// Mitsubishi GX Works2 project: plc 기말 신호등   PLC: Q02/Q02H

PROGRAM MAIN
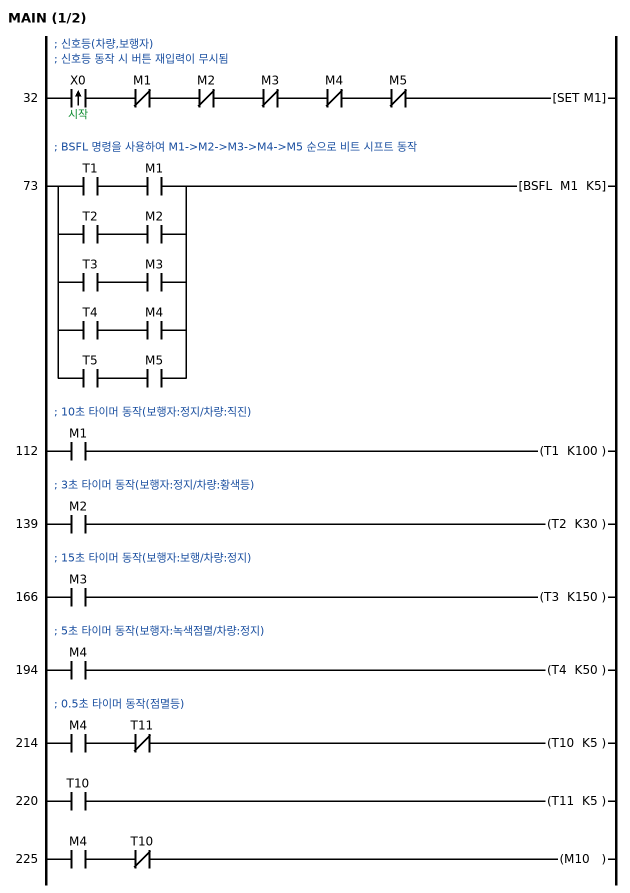
; 신호등(차량,보행자)
; 신호등 동작 시 버튼 재입력이 무시됨
32    LDP     X0  ; 시작
      ANI     M1
      ANI     M2
      ANI     M3
      ANI     M4
      ANI     M5
      SET     M1
; BSFL 명령을 사용하여 M1->M2->M3->M4->M5 순으로 비트 시프트 동작
73    LD      T1
      AND     M1
      LD      T2
      AND     M2
      ORB
      LD      T3
      AND     M3
      ORB
      LD      T4
      AND     M4
      ORB
      LD      T5
      AND     M5
      ORB
      BSFL    M1 K5
; 10초 타이머 동작(보행자:정지/차량:직진)
112   LD      M1
      OUT     T1 K100
; 3초 타이머 동작(보행자:정지/차량:황색등)
139   LD      M2
      OUT     T2 K30
; 15초 타이머 동작(보행자:보행/차량:정지)
166   LD      M3
      OUT     T3 K150
; 5초 타이머 동작(보행자:녹색점멸/차량:정지)
194   LD      M4
      OUT     T4 K50
; 0.5초 타이머 동작(점멸등)
214   LD      M4
      ANI     T11
      OUT     T10 K5
220   LD      T10
      OUT     T11 K5
225   LD      M4
      ANI     T10
      OUT     M10
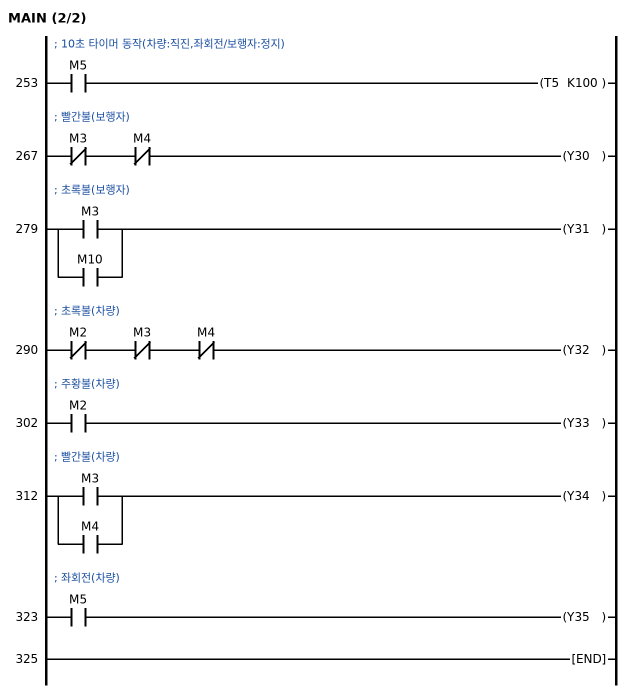
; 10초 타이머 동작(차량:직진,좌회전/보행자:정지)
253   LD      M5
      OUT     T5 K100
; 빨간불(보행자)
267   LDI     M3
      ANI     M4
      OUT     Y30
; 초록불(보행자)
279   LD      M3
      OR      M10
      OUT     Y31
; 초록불(차량)
290   LDI     M2
      ANI     M3
      ANI     M4
      OUT     Y32
; 주황불(차량)
302   LD      M2
      OUT     Y33
; 빨간불(차량)
312   LD      M3
      OR      M4
      OUT     Y34
; 좌회전(차량)
323   LD      M5
      OUT     Y35
325   END
END_PROGRAM
